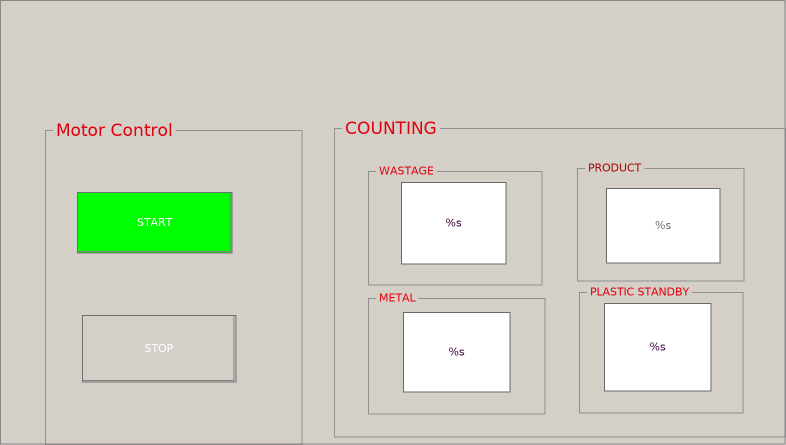
VISUALIZATION Visualization  // 786x445
    GroupBox (45,122 257x323), "Motor Control"
        Button (32,70 155x61), "START", text variable: GVL.start
        Button (37,193 154x67), "STOP", text variable: GVL.stop
    GroupBox (334,120 452x317), "COUNTING"
        GroupBox (34,43 174x122), "WASTAGE"
            Textfield (33,19 105x82), "%s", text variable: MAIN.Wastage
        GroupBox (243,40 167x121), "PRODUCT"
            Textfield (29,28 114x75), "%s", text variable: MAIN.FinalProduct
        GroupBox (34,170 177x124), "METAL"
            Textfield (35,22 107x80), "%s", text variable: MAIN.MetalCount
        GroupBox (245,164 164x129), "PLASTIC STANDBY"
            Textfield (25,19 107x88), "%s", text variable: MAIN.Plactic_Count
END_VISUALIZATION

(* stored: Version 1.1.0.1, ProductVersion 3.1.4024.12
   Visu Visualization: Id {6c2320c8-3b9d-4573-acfb-3c2178bdef00} *)
